// TwinCAT 3 PLC project Untitled1
// ProgramVersion: 3.1.4026.1+c9eadab3edd020c56c333d811d5b3c408c2550c8
// libraries:
//   Tc2_Standard, * (Beckhoff Automation GmbH)
//   Tc2_System, * (Beckhoff Automation GmbH)
// project tree:
//   PLC Command/Deco/ F_Deco.TcPOU, PRG_DecoSample.TcPOU
//   PLC Command/Move/ PRG_Move.TcPOU
//   / PlcTask.TcTTO
//   POUs/ MAIN.TcPOU
// real-time tasks:
//   TASK PlcTask: cycle T#10ms, priority 20, ADS port 350

CONFIGURATION Untitled1
    RESOURCE PLC ON TwinCAT3
        TASK PlcTask(INTERVAL := T#10ms, PRIORITY := 20);
        PROGRAM MAIN WITH PlcTask : MAIN;
    END_RESOURCE
END_CONFIGURATION

// ---- POUs/MAIN.TcPOU
PROGRAM MAIN
VAR
END_VAR

PRG_DecoSample();
PRG_MOVE();

END_PROGRAM

// ---- PLC Command/Deco/PRG_DecoSample.TcPOU
PROGRAM PRG_DecoSample
VAR
	(* Deco 기능 테스트 *)
	nWord_test1 : DWORD;
	nWord_test2 : DWORD;
	nWord_test3 : DWORD;
	//마우스 우클릭 => Display mode => Binary 선택시 온라인값 이진수로 확인가능 
END_VAR

nWord_Test1 := F_Deco(1); //1번째 비트 TRUE
nWord_Test2 := F_Deco(5); //5번째 비트 TRUE
nWord_Test3 := F_Deco(31);//31번째 비트 TRUE

END_PROGRAM

// ---- PLC Command/Deco/F_Deco.TcPOU
FUNCTION F_Deco : DWORD
VAR_INPUT
	DecoIn : UINT;
END_VAR

CASE DecoIn OF
	1: F_Deco.0 := TRUE;
	2: F_Deco.1 := TRUE;
	3: F_Deco.2 := TRUE;
	4: F_Deco.3 := TRUE;
	5: F_Deco.4 := TRUE;
	6: F_Deco.5 := TRUE;
	7: F_Deco.6 := TRUE;
	8: F_Deco.7 := TRUE;
	9: F_Deco.8 := TRUE;
	10:F_Deco.9 := TRUE;
	11:F_Deco.10:= TRUE;
	12:F_Deco.11:= TRUE;
	13:F_Deco.12:= TRUE;
	14:F_Deco.13:= TRUE;
	15:F_Deco.14:= TRUE;
	16:F_Deco.15:= TRUE;
	17:F_Deco.16:= TRUE;
	18:F_Deco.17:= TRUE;
	19:F_Deco.18:= TRUE;
	20:F_Deco.19:= TRUE;
	21:F_Deco.20 := TRUE;
	22:F_Deco.21 := TRUE;
	23:F_Deco.22 := TRUE;
	24:F_Deco.23 := TRUE;
	25:F_Deco.24 := TRUE;
	26:F_Deco.25 := TRUE;
	27:F_Deco.26 := TRUE;
	28:F_Deco.27 := TRUE;
	29:F_Deco.28 := TRUE;
	30:F_Deco.29 := TRUE;
	31:F_Deco.30 := TRUE;
	32:F_Deco.31 := TRUE;
	ELSE
		RETURN;
END_CASE

END_FUNCTION

// ---- PLC Command/Move/PRG_Move.TcPOU
PROGRAM PRG_Move
VAR
	var1 : INT := 11;
	var2 : INT := 20;
	
	var3 : INT := 11;
	var4 : INT := 30;
END_VAR

var2 := MOVE(var1);
var4 := var3;

END_PROGRAM
